FUNCTION_BLOCK FB_CylinderDiag EXTENDS FB_CylinderBase
VAR_INPUT
	nTimeOut						:		TIME;			// Watchdog time for cylinder position monitoring
END_VAR
VAR_OUTPUT
	bError						:		BOOL;			// Error signal (derived from position watchdog)
	nErrorID					:		UDINT;			// Error ID
	sErrorMsg					:		STRING;			// Error Message
END_VAR
VAR
	fbTriggerError				:		R_TRIG;			// Trigger to recognize rising edge of error
	fbTimerWatchDog				:		TON;			// Watchdog timer for monitoring if cylinder reaches base/work position
END_VAR

// ============================================================
;
// ============================================================

METHOD Diag
VAR_INPUT
END_VAR
IF NOT bAtBasePos AND NOT bAtWorkPos THEN
	fbTimerWatchDog(	IN		:=		TRUE,
						PT		:=		nTimeOut);
ELSE
	fbTimerWatchDog(	IN		:=		FALSE,
						PT		:=		nTimeOut);
END_IF

	fbTriggerError(		CLK		:=		fbTimerWatchDog.Q);
	
	bError						:=		fbTimerWatchDog.Q;
	
IF bError	THEN
	IF	bMoveToWork		THEN
		sErrorMsg		:=		'Work position not reached';
		nErrorID		:=		92;
	ELSE
		sErrorMsg		:=		'Base position not reached';
		nErrorID		:=		91;
	END_IF
ELSE
	sErrorMsg			:=		'';
	nErrorID			:=		0;
END_IF
END_METHOD

METHOD Reset

// Calling Reset() method of parental class FB_Cylinder
SUPER^.Reset();

bError			:=		FALSE;
nErrorID		:=		0;
sErrorMsg		:=		'';
END_METHOD

METHOD PROTECTED StateMachine
VAR_INPUT
	bBasePosReq		:	BOOL;
	bWorkPosReq		:	BOOL;
END_VAR
IF NOT bError THEN
	// Calling StateMachine() method of parental class FB_Cylinder
	SUPER^.StateMachine(	bBasePosReq			:=		bBasePosReq,
							bWorkPosReq			:=		bWorkPosReq);
	
	// Diagnosis evaluation by every movement of cylinder							
	Diag();
END_IF
END_METHOD

END_FUNCTION_BLOCK

(* stored: Version 1.1.0.1, ProductVersion 3.1.4024.15
   POU FB_CylinderDiag: Id {27692f1f-fa73-43e8-89a4-19c70e80f4d6}, SpecialFunc None
   Method Diag: Id {23328d7b-9ce9-4e2c-bca7-2ce8214bd706}
   Method Reset: Id {0f5a6a7f-9ace-41fc-a5c4-04b5518e128c}
   Method StateMachine: Id {371d7597-83fb-4be1-ba55-f2eecf674496} *)
